ABB RobotStudio station: EstaciónFinal.rspag

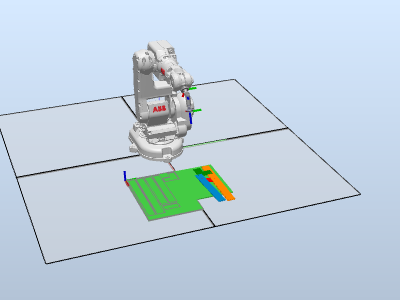
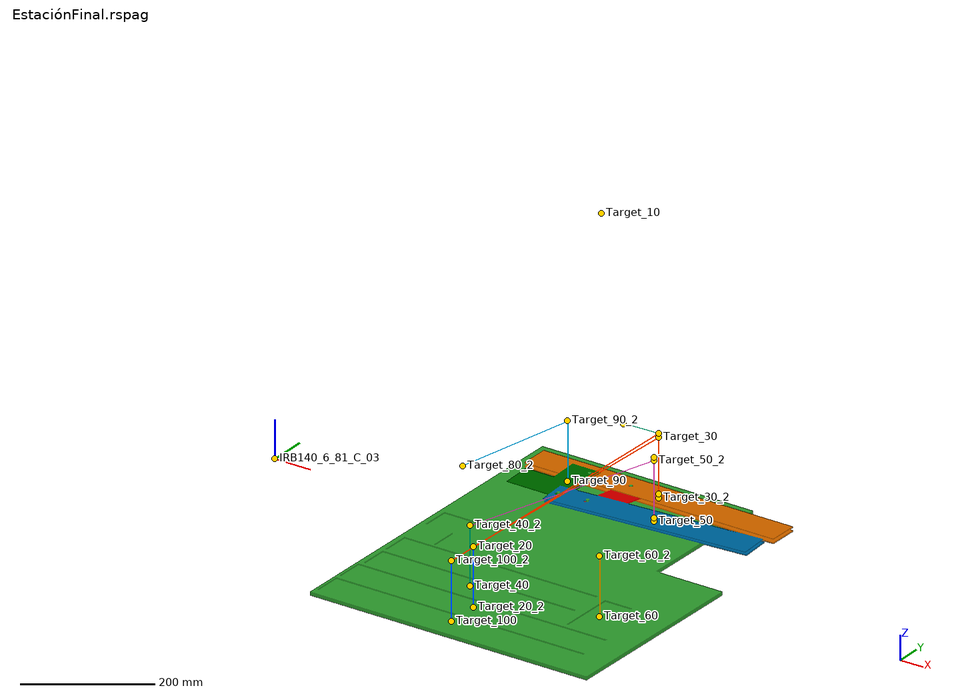
[picture v1: parts stored in the station drawn from their meshes, with robot base, taught points and paths (robot models come from the ABB library and are not in the file)]
--- station ---
Station Estación (saved by RobotStudio 22.2.9947.0)
Controller IRB140_6_81
  mechanical unit ROB_1: IRB140_6_81_C_03, 6 joints, base frame (0, 0, 0) mm
Layout (positions relative to the parent item):
  - IRB140_6_81_C_03 [mechanism, from Robots\IRB140_6_81_C_G_03.rslib] at (0, 0, 0) mm; joint values [0, 0, 0, 0, 0.5236, 0] (rad or m)
  - Ventosa [mechanism] at (506.29, 0, 679.5) mm, rotated rx -180 ry 60 rz -180 deg
      TCP succión at (53.19, 0, 127.26) mm, rotated rx 0 ry 40 rz 0 deg
      links: HerramientaAlineada
  - LineSensor [smart component, from Components\LineSensor.rslib] at (589.91, 0, 569.81) mm, rotated rx -180 ry 20 rz -180 deg
      properties: Start=[0 0 -0.002]; End=[0 0 0.002]; Radius=0.002; SensedPart=(none); SensedPoint=[0 0 0]
    - _sensorPart_ [part], size 4 x 4 x 4 mm
  - Attacher [smart component, from Components\Attacher.rslib]
      properties: Parent=Ventosa; Flange=0; Child=(none); Mount=false; Offset=[0 0 0]; Orientation=[0 0 0]
  - Detacher [smart component, from Components\Detacher.rslib]
      properties: Child=(none); KeepPosition=true
  - ConjuntoDeEnsamble [part] at (743.64, 25.69, 0) mm, size 500 x 600 x 16 mm
  - Pinz [part] at (414.58, 164.52, 12.04) mm, rotated rx 89.2 ry 1.41 rz -89 deg, size 100 x 2 x 100 mm
  - Lup [part] at (551.12, 203.82, 8) mm, rotated rx -90 ry 0 rz 90 deg, size 50 x 2 x 450 mm
  - Lup_2 [part] at (550.6, 204.5, 8) mm, rotated rx -90 ry 0 rz 90 deg, size 50 x 2 x 450 mm
  - Ldw [part] at (590.34, 136, 8) mm, rotated rx -90 ry 0 rz 94 deg, size 50 x 2 x 350 mm
  - Ldw_2 [part] at (590.34, 136, 8) mm, rotated rx -90 ry 0 rz 94 deg, size 50 x 2 x 350 mm
  - Borde [part] at (743.64, 25.69, 0) mm, size 500 x 350 x 0 mm
  - Pinz_2 [part] at (411, 164.5, 11) mm, rotated rx 90 ry 0 rz -90 deg, size 100 x 2 x 100 mm
  - H [part] at (503.29, 164.41, 11.96) mm, rotated rx -91.15 ry 1.13 rz 163.97 deg, size 50 x 2 x 100 mm
  - H_2 [part] at (503, 162, 11) mm, rotated rx -90 ry 0 rz 162 deg, size 50 x 2 x 100 mm
  - Ldw_3 [part] at (590.58, 132.69, 13.84) mm, rotated rx -90 ry 0 rz 94 deg, size 50 x 2 x 350 mm
  - Lup_3 [part] at (550.6, 204.5, 14) mm, rotated rx -90 ry 0 rz 90 deg, size 50 x 2 x 450 mm
  - Lup_4 [part] at (550.6, 204.5, 14) mm, rotated rx -90 ry 0 rz 90 deg, size 50 x 2 x 450 mm
  - Ldw_4 [part] at (590.34, 136, 14) mm, rotated rx -90 ry 0 rz 94 deg, size 50 x 2 x 350 mm
  - LogicGate [smart component, from Components\LogicGate.rslib]
      properties: Operator=NOT; Delay=0
  - Positioner_H [smart component, from Components\Positioner.rslib]
      properties: Object=H; Position=[0.7053 -0.1685 0.005]; Orientation=[-1.5707963267949 0 3.14159265358979]; Reference=Global; ReferenceObject=(none)
  - Positioner_Pinz [smart component, from Components\Positioner.rslib]
      properties: Object=Pinz; Position=[0.3645 -0.0363 0.003]; Orientation=[1.5707963267949 0 0]; Reference=Global; ReferenceObject=(none)
  - Positioner_Lup [smart component, from Components\Positioner.rslib]
      properties: Object=Lup; Position=[0.53474 -0.25139 0.005]; Orientation=[-1.5707963267949 0 1.5707963267949]; Reference=Global; ReferenceObject=(none)
  - Positioner_Lup_3 [smart component, from Components\Positioner.rslib]
      properties: Object=Lup_3; Position=[0.53474 -0.30851 0.005]; Orientation=[-1.5707963267949 0 1.5707963267949]; Reference=Global; ReferenceObject=(none)
  - Positioner_Ldw [smart component, from Components\Positioner.rslib]
      properties: Object=Ldw; Position=[0.48934 -0.19539 0.005]; Orientation=[-1.5707963267949 0 1.5707963267949]; Reference=Global; ReferenceObject=(none)
  - Positioner_Ldw_3 [smart component, from Components\Positioner.rslib]
      properties: Object=Ldw_3; Position=[0.48934 -0.13879 0.005]; Orientation=[-1.5707963267949 0 1.5707963267949]; Reference=Global; ReferenceObject=(none)
Attachment: Ventosa is attached to IRB140_6_81_C_03 / Link6
Attachment: LineSensor is attached to Ventosa / HerramientaAlineada
Station signals: DI PH
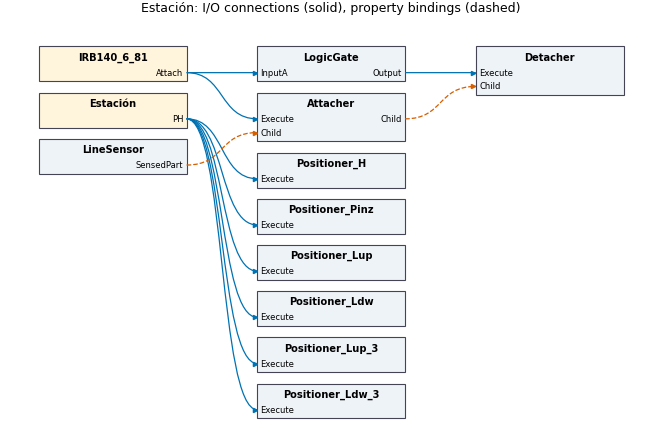
Station logic (signal -> signal, property => property):
  IRB140_6_81.Attach -> Attacher.Execute
  IRB140_6_81.Attach -> LogicGate.InputA
  LogicGate.Output -> Detacher.Execute
  Estación.PH -> Positioner_H.Execute
  Estación.PH -> Positioner_Pinz.Execute
  Estación.PH -> Positioner_Lup.Execute
  Estación.PH -> Positioner_Ldw.Execute
  Estación.PH -> Positioner_Lup_3.Execute
  Estación.PH -> Positioner_Ldw_3.Execute
  LineSensor.SensedPart => Attacher.Child
  Attacher.Child => Detacher.Child

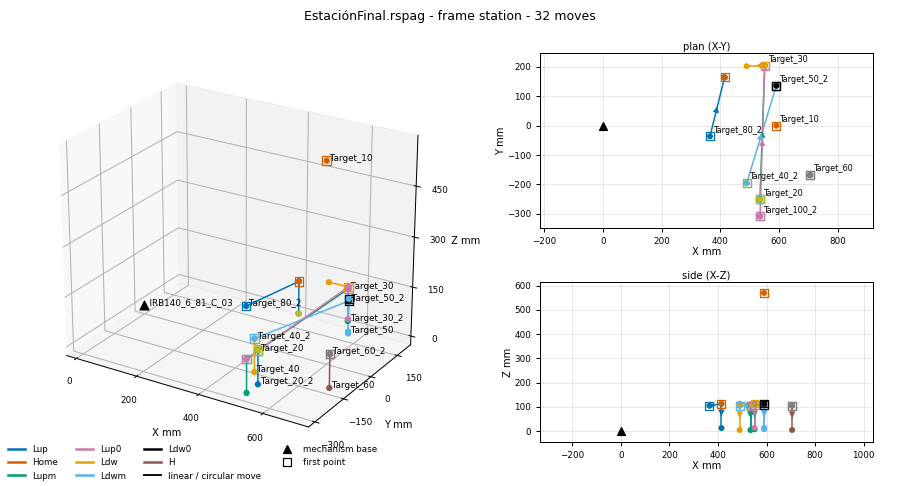
[picture p0: tool path of EstaciónFinal.rspag in frame station, 32 of 46 moves have a stored position in this frame; points joined in program order, loops and branches not executed]
--- Backups/IRB140_6_81/RAPID/TASK1/PROGMOD/CalibData.mod ---
MODULE CalibData
    PERS tooldata succión:=[TRUE,[[53.19,0,127.26],[0.939692621,0,0.342020143,0]],[1,[15.567,0,59.596],[1,0,0,0],0,0,0]];
    TASK PERS wobjdata Tabla:=[FALSE,TRUE,"",[[0,0,0],[1,0,0,0]],[[305.640809361,-345.526,4.80199935],[0.999935152,0.011259768,-0.001705395,0.000019204]]];
ENDMODULE

--- Backups/IRB140_6_81/RAPID/TASK1/PROGMOD/Module1.mod ---
MODULE Module1
    CONST robtarget Target_20:=[[229.12374666,96.731764507,97.263749646],[0.0045   ,-0.7009    ,0.7132   ,-0.0105],[-1,0,-2,0],[9E+09,9E+09,9E+09,9E+09,9E+09,9E+09]];
    CONST robtarget Target_20_2:=[[228.782590129,94.479925502,-2.710311156],[0.005884839,0.38264087,-0.923826969,0.00975011],[-1,0,-2,0],[9E+09,9E+09,9E+09,9E+09,9E+09,9E+09]];
    CONST robtarget Target_10:=[[286.192182184,358.139537963,556.107701921],[0.171957146,-0.001936356,0.985040077,-0.011092229],[0,0,0,0],[9E+09,9E+09,9E+09,9E+09,9E+09,9E+09]];
    CONST robtarget Target_30:=[[245.510885963,551.88763337,89.95657104],[0.005884839,0.38264087,-0.923826969,0.00975011],[0,1,-2,0],[9E+09,9E+09,9E+09,9E+09,9E+09,9E+09]];
    CONST robtarget Target_30_2:=[[245.169729432,549.635794365,-10.017489763],[0.005884839,0.38264087,-0.923826969,0.00975011],[0,1,-2,0],[9E+09,9E+09,9E+09,9E+09,9E+09,9E+09]];
    CONST robtarget Target_40_2:=[[184.040008961,152.340124362,96.165060034],[0.005884839,0.38264087,-0.923826969,0.00975011],[-1,1,-2,0],[9E+09,9E+09,9E+09,9E+09,9E+09,9E+09]];
    CONST robtarget Target_40:=[[183.69885248,150.088285465,-3.809000771],[0.005884839,0.38264087,-0.923826969,0.00975011],[-1,1,-2,0],[9E+09,9E+09,9E+09,9E+09,9E+09,9E+09]];
    CONST robtarget Target_50_2:=[[285.049655836,483.705888558,91.357388428],[0.006221193,0.414648876,-0.909910226,0.009538737],[0,0,-2,0],[9E+09,9E+09,9E+09,9E+09,9E+09,9E+09]];
    CONST robtarget Target_50:=[[284.708443179,481.45404643,-8.616762357],[0.006221193,0.414648876,-0.909910226,0.009538737],[0,1,-2,0],[9E+09,9E+09,9E+09,9E+09,9E+09,9E+09]];
    CONST robtarget Target_60_2:=[[400.096751677,179.051746899,94.826118299],[0.005884839,0.38264087,-0.923826969,0.00975011],[-1,0,-1,0],[9E+09,9E+09,9E+09,9E+09,9E+09,9E+09]];
    CONST robtarget Target_60:=[[399.755595146,176.799907894,-5.147942503],[0.005884839,0.38264087,-0.923826969,0.00975011],[-1,0,-2,0],[9E+09,9E+09,9E+09,9E+09,9E+09,9E+09]];
    CONST robtarget Target_70_2:=[[197.720398886,509.773560591,94.069019261],[0.004287134,0.233411549,-0.972311346,0.010550662],[0,-1,0,1],[9E+09,9E+09,9E+09,9E+09,9E+09,9E+09]];
    CONST robtarget Target_70:=[[197.37924231,507.521721572,-5.905041541],[0.004287134,0.233411549,-0.972311346,0.010550662],[0,-1,0,1],[9E+09,9E+09,9E+09,9E+09,9E+09,9E+09]];
    CONST robtarget Target_80_2:=[[59.200735476,311.399373985,93.008380327],[0.011259958,0.99993515,-0.000019207,-0.001705677],[-1,1,-1,1],[9E+09,9E+09,9E+09,9E+09,9E+09,9E+09]];
    CONST robtarget Target_80:=[[58.859578945,309.14753498,-6.965680475],[0.011259958,0.99993515,-0.000019207,-0.001705677],[-1,1,-1,1],[9E+09,9E+09,9E+09,9E+09,9E+09,9E+09]];
    CONST robtarget Target_90_2:=[[108.933738622,512.046855311,96.321314041],[0.009168088,0.707047344,-0.707074507,0.006755897],[0,-2,0,1],[9E+09,9E+09,9E+09,9E+09,9E+09,9E+09]];
    CONST robtarget Target_90:=[[108.592582168,509.795016351,-3.652746763],[0.009168088,0.707047343,-0.707074507,0.006755897],[0,0,-2,0],[9E+09,9E+09,9E+09,9E+09,9E+09,9E+09]];
    CONST robtarget Target_100_2:=[[229.439744782,39.245320884,98.557509349],[0.005884839,0.38264087,-0.923826969,0.00975011],[-1,0,-2,0],[9E+09,9E+09,9E+09,9E+09,9E+09,9E+09]];

    CONST robtarget Target_100:=[[229.098588301,36.993481987,-1.416551456],[0.005884839,0.38264087,-0.923826969,0.00975011],[-1,0,-2,0],[9E+09,9E+09,9E+09,9E+09,9E+09,9E+09]];
    CONST robtarget Target_110_2:=[[245.330356475,552.326681957,95.94885461],[0.005884839,0.38264087,-0.923826969,0.00975011],[0,1,-2,0],[9E+09,9E+09,9E+09,9E+09,9E+09,9E+09]];

    CONST robtarget Target_110:=[[244.989199994,550.07484306,-4.025206195],[0.005884839,0.38264087,-0.923826969,0.00975011],[0,1,-2,0],[9E+09,9E+09,9E+09,9E+09,9E+09,9E+09]];
    CONST robtarget Target_110_1_1:=[[183.69885247,550.07484306,95.94885461],[0.005884839,0.38264087,-0.923826969,0.00975011],[0,1,-2,0],[9E+09,9E+09,9E+09,9E+09,9E+09,9E+09]];
    CONST robtarget Target_110_1_2:=[[183.69,550.0-320-15-5,95],[0.005884839,0.38264087,-0.923826969,0.00975011],[0,1,-2,0],[9E+09,9E+09,9E+09,9E+09,9E+09,9E+09]];
    CONST robtarget Target_110_1_3:=[[183.69,550.0-320-15-5,-5],[0.005884839,0.38264087,-0.923826969,0.00975011],[0,1,-2,0],[9E+09,9E+09,9E+09,9E+09,9E+09,9E+09]];
    CONST robtarget Target_110_1_4:=[[183.69,550.0-320-15-5,95],[0.005884839,0.38264087,-0.923826969,0.00975011],[0,1,-2,0],[9E+09,9E+09,9E+09,9E+09,9E+09,9E+09]];

    CONST robtarget Target_120_2:=[[183.69885247,206.673933174,94.89051174],[0.005884839,0.38264087,-0.923826969,0.00975011],[-1,0,2,0],[9E+09,9E+09,9E+09,9E+09,9E+09,9E+09]];
    CONST robtarget Target_120:=[[183.69885247,206.673933174,-5.083549065],[0.005884839,0.38264087,-0.923826969,0.00975011],[-1,1,2,0],[9E+09,9E+09,9E+09,9E+09,9E+09,9E+09]];

    CONST robtarget Target_130_2:=[[285.070125228,483.840998898,97.355832076],[0.006221193,0.414648876,-0.909910226,0.009538737],[0,0,-2,0],[9E+09,9E+09,9E+09,9E+09,9E+09,9E+09]];
    CONST robtarget Target_130:=[[284.728909186,481.589154491,-2.618318646],[0.006221193,0.414648876,-0.909910226,0.009538737],[0,1,-2,0],[9E+09,9E+09,9E+09,9E+09,9E+09,9E+09]];

    CONST robtarget Target_60_3:=[[400.096751677-200+20,179.051746899+150,94.826118299],[0.0091   ,-0.2503    ,0.9681   ,-0.0068],[-1,0,-1,0],[9E+09,9E+09,9E+09,9E+09,9E+09,9E+09]];
    CONST robtarget Target_60_4:=[[197.720398886-40+5+35,509.773560591+10-10,94.069019261],[0.0091   ,-0.2503    ,0.9681   ,-0.0068],[0,0,-1,0],[9E+09,9E+09,9E+09,9E+09,9E+09,9E+09]];
    CONST robtarget Target_60_5:=[[197.720398886-40+5+35,509.773560591+10-10,-5],[0.0091   ,-0.2503    ,0.9681   ,-0.0068],[0,0,-1,0],[9E+09,9E+09,9E+09,9E+09,9E+09,9E+09]];
    CONST robtarget Target_60_6:=[[197.720398886-40+5+35,509.773560591+10-10,94.069019261],[0.0091   ,-0.2503    ,0.9681   ,-0.0068],[0,0,-1,0],[9E+09,9E+09,9E+09,9E+09,9E+09,9E+09]];

    CONST robtarget Target_20_1:=[[229.12374666,96.731764507+250,97.263749646],[0.0045   ,-0.7009    ,0.7132   ,-0.0105],[-1,0,-2,0],[9E+09,9E+09,9E+09,9E+09,9E+09,9E+09]];

    CONST robtarget Target_80_2_1:=[[229.12374666-200,96.731764507+200,97.263749646],[0.0042    ,0.9999   ,-0.0087    ,0.0106],[-1,0,-2,0],[9E+09,9E+09,9E+09,9E+09,9E+09,9E+09]];
    !CONST robtarget Target_80_2_2:=[[229.12374666-200,96.731764507+250,97.263749646],[0.0042    ,0.9999   ,-0.0087    ,0.0106],[-1,0,-2,0],[9E+09,9E+09,9E+09,9E+09,9E+09,9E+09]];
    CONST robtarget Target_80_2_3:=[[49.1237+10,311.7318-3,97.263749646],[0.0042    ,0.9999   ,-0.0087    ,0.0106],[-1,0,-2,0],[9E+09,9E+09,9E+09,9E+09,9E+09,9E+09]];
    CONST robtarget Target_80_2_4:=[[49.1237+10,  311.7318-3,-8.0],[0.0042    ,0.9999   ,-0.0087    ,0.0106],[-1,0,-2,0],[9E+09,9E+09,9E+09,9E+09,9E+09,9E+09]];
    !CONST robtarget Target_80_3:=[[59.200735476,311.399373985,93.008380327],[0.011259958,0.99993515,-0.000019207,-0.001705677],[-1,1,-1,1],[9E+09,9E+09,9E+09,9E+09,9E+09,9E+09]];
    !CONST robtarget Target_120_2:=[[184.040008951,208.925772071,94.89051174],[0.005884839,0.38264087,-0.923826969,0.00975011],[-1,0,2,0],[9E+09,9E+09,9E+09,9E+09,9E+09,9E+09]];
    CONST robtarget Target_80_2_5:=[[49.1237+65,  311.7318+220,97.263749646],[0.0045   ,-0.7009    ,0.7132   ,-0.0105],[-1,0,-2,0],[9E+09,9E+09,9E+09,9E+09,9E+09,9E+09]];
    CONST robtarget Target_80_2_6:=[[49.1237+65,  311.7318+220,-11],[0.0045   ,-0.7009    ,0.7132   ,-0.0105],[-1,0,-2,0],[9E+09,9E+09,9E+09,9E+09,9E+09,9E+09]];
    CONST robtarget Target_80_2_7:=[[49.1237+65,  311.7318+220,97.263749646],[0.0045   ,-0.7009    ,0.7132   ,-0.0105],[-1,0,-2,0],[9E+09,9E+09,9E+09,9E+09,9E+09,9E+09]];

    CONST robtarget Target_90_2_1:=[[108.933738622,512.046855311,96.321314041],[0.0045   ,-0.7009    ,0.7132   ,-0.0105],[0,-2,0,1],[9E+09,9E+09,9E+09,9E+09,9E+09,9E+09]];
    CONST robtarget Target_90_1:=[[108.592582168,509.795016351,-3.652746763],[0.0045   ,-0.7009    ,0.7132   ,-0.0105],[0,-2,0,1],[9E+09,9E+09,9E+09,9E+09,9E+09,9E+09]];

    CONST intnum t := 1;

    PROC main()
        SetDO Attach,0;
        Home;
        Lup;
        WaitTime(t);
        SetDO Attach,1;
        WaitTime(t);
        Lupm;
        WaitTime(t);
        SetDO Attach,0;
        WaitTime(t);
        Lup0;
        Ldw;
        WaitTime(t);
        SetDO Attach,1;
        WaitTime(t);
        Ldwm;
        WaitTime(t);
        SetDO Attach,0;
        WaitTime(t);
        Ldw0;
        H;
        WaitTime(t);
        SetDO Attach,1;
        WaitTime(t);
        Hm;
        H0;
        L;
        Lup3;
        WaitTime(t);
        SetDO Attach,1;
        WaitTime(t);
        Lup3m;
        WaitTime(t);
        SetDO Attach,0;
        WaitTime(t);
        Lup30;
        Ldw3;
        Ldw3m;
        WaitTime(t);
        SetDO Attach,0;
        WaitTime(t);
        Ldw30;
        Home;
        SetDO Attach,0;
    ENDPROC

    PROC Lup()
        MoveL Target_20,v200,z30,succión\WObj:=Tabla;
        MoveL Target_20_2,v200,z30,succión\WObj:=Tabla;
    ENDPROC
    PROC Home()
        MoveL Target_10,v200,z30,succión\WObj:=Tabla;
    ENDPROC
    PROC Lupm()
        MoveL Target_20,v200,z30,succión\WObj:=Tabla;
        MoveL Target_30,v200,z30,succión\WObj:=Tabla;
        MoveL Target_30_2,v200,z30,succión\WObj:=Tabla;
    ENDPROC
    PROC Lup0()
        MoveL Target_30,v200,z30,succión\WObj:=Tabla;
    ENDPROC
    PROC Ldw()
        MoveL Target_40_2,v200,z30,succión\WObj:=Tabla;
        MoveL Target_40,v200,z30,succión\WObj:=Tabla;
    ENDPROC
    PROC Ldwm()
        MoveL Target_40_2,v200,z30,succión\WObj:=Tabla;
        MoveL Target_50_2,v200,z30,succión\WObj:=Tabla;
        MoveL Target_50,v200,z30,succión\WObj:=Tabla;
    ENDPROC
    PROC Ldw0()
        MoveL Target_50_2,v200,z30,succión\WObj:=Tabla;
    ENDPROC
    PROC H()
        MoveL Target_60_2,v200,z30,succión\WObj:=Tabla;
        MoveL Target_60,v200,z30,succión\WObj:=Tabla;

    ENDPROC
    PROC Hm()
        MoveL Target_60_2,v200,z30,succión\WObj:=Tabla;
        MoveL Target_60_3,v200,z30,succión\WObj:=Tabla;
        MoveL Target_60_4,v200,z30,succión\WObj:=Tabla;
        MoveL Target_60_5,v200,z30,succión\WObj:=Tabla;
        WaitTime(t);
        SetDO Attach,0;
        WaitTime(t);
        MoveL Target_60_6,v200,z30,succión\WObj:=Tabla;

    ENDPROC
    PROC H0()
        !MoveL Target_70_2,v200,z30,succión\WObj:=Tabla;
    ENDPROC
    PROC L()
        MoveL Target_20,v200,z30,succión\WObj:=Tabla;
        MoveL Target_20_1,v200,z30,succión\WObj:=Tabla;
        MoveL Target_80_2_1,v200,z30,succión\WObj:=Tabla;
        MoveL Target_80_2_3,v200,z30,succión\WObj:=Tabla;
        MoveL Target_80_2_4,v200,z30,succión\WObj:=Tabla;
        WaitTime(t);
        SetDO Attach,1;
        WaitTime(t);
        MoveL Target_80_2_3,v200,z30,succión\WObj:=Tabla;
        !Bajar y
        MoveL Target_80_2_5,v200,z30,succión\WObj:=Tabla;
        !yo MoveL Target_80_2_6,v200,z30,succión\WObj:=Tabla;
        MoveL Target_90,v200,z30,succión\WObj:=Tabla;
        WaitTime(t);
        SetDO Attach,0;
        WaitTime(t);
        MoveL Target_80_2_7,v200,z30,succión\WObj:=Tabla;

    ENDPROC
    PROC Lm()
        MoveL Target_80_2,v200,z30,succión\WObj:=Tabla;
        MoveL Target_90_2,v200,z30,succión\WObj:=Tabla;
        MoveL Target_90,v200,z30,succión\WObj:=Tabla;
    ENDPROC
    PROC L0()
        MoveL Target_90_2,v200,z30,succión\WObj:=Tabla;
    ENDPROC
    PROC Lup3()
        MoveL Target_100_2,v200,z30,succión\WObj:=Tabla;
        MoveL Target_100,v200,z30,succión\WObj:=Tabla;
    ENDPROC
    PROC Lup3m()
        MoveL Target_100_2,v200,z30,succión\WObj:=Tabla;
        MoveL Target_110_2,v200,z30,succión\WObj:=Tabla;
        MoveL Target_110,v200,z30,succión\WObj:=Tabla;

    ENDPROC
    PROC Lup30()
        MoveL Target_110_2,v200,z30,succión\WObj:=Tabla;
        MoveL Target_110_1_1,v200,z30,succión\WObj:=Tabla;
        MoveL Target_110_1_2,v200,z30,succión\WObj:=Tabla;
        MoveL Target_110_1_3,v200,z30,succión\WObj:=Tabla;
        WaitTime(t);
        SetDO Attach,1;
        WaitTime(t);
        MoveL Target_110_1_4,v200,z30,succión\WObj:=Tabla;
        !MoveL Target_120_2,v200,z30,succión\WObj:=Tabla;
        !MoveL Target_120,v200,z30,succión\WObj:=Tabla;
    ENDPROC
    PROC Ldw3()

    ENDPROC
    PROC Ldw3m()
        MoveL Target_130_2,v200,z30,succión\WObj:=Tabla;
        MoveL Target_130,v200,z30,succión\WObj:=Tabla;
    ENDPROC
    PROC Ldw30()
        MoveL Target_130_2,v200,z30,succión\WObj:=Tabla;
    ENDPROC
ENDMODULE

--- Backups/IRB140_6_81/SYSPAR/EIO.cfg ---
EIO:CFG_1.0:6:1::
#
EIO_SIGNAL:

      -Name "Attach" -SignalType "DO"
